// TwinCAT 3 PLC project PLC1
// ProgramVersion: 3.1.4024.0
// libraries:
//   Tc2_Standard, * (Beckhoff Automation GmbH)
//   Tc2_System, * (Beckhoff Automation GmbH)
//   Tc3_Module, * (Beckhoff Automation GmbH)
// project tree:
//   DUTs/ machineStates.TcDUT
//   / PlcTask.TcTTO
//   POUs/ DOSomething.TcPOU, MAIN.TcPOU
// real-time tasks:
//   TASK PlcTask: cycle T#10ms, priority 20, ADS port 350

CONFIGURATION PLC1
    RESOURCE PLC ON TwinCAT3
        TASK PlcTask(INTERVAL := T#10ms, PRIORITY := 20);
        PROGRAM MAIN WITH PlcTask : MAIN;
    END_RESOURCE
END_CONFIGURATION

// ---- DUTs/machineStates.TcDUT
{attribute 'qualified_only'}
{attribute 'strict'}
TYPE machineStates :
(
	START_OF_DAY,
	DURING_DAY,
	END_OF_DAY,
	DISARMED
);
END_TYPE

// ---- POUs/MAIN.TcPOU
PROGRAM MAIN
VAR
	doSomething_instance1: DoSomething;
	
END_VAR

doSomething_instance1.method1();
doSomething_instance1(input := true);

END_PROGRAM

// ---- POUs/DOSomething.TcPOU
FUNCTION_BLOCK DOSomething
VAR_INPUT
	input :BOOL;
END_VAR
VAR_OUTPUT
END_VAR
VAR
	isDoorOpen : BOOL;
END_VAR

IF isDoorOpen THEN
	//
END_IF

METHOD method1 : BOOL
VAR_INPUT
END_VAR
VAR
	currentAlarm1State : machineStates;
	currentAlarm2State : machineStates;
END_VAR
//do something
case
END_METHOD

END_FUNCTION_BLOCK
